// TIA Portal V20 export
DATA_BLOCK "Config"   // DB100
// stored: MemoryReserve 100, Namespace Unit1.Em7
   VAR
      em : "LAF_typeEmConfiguration";   // Configuration of EM Parameters
      axis : Array[1.._.U1EM7_NO_OF_AXES] of DB_ANY;
      cam : Array[1.._.U1EM7_NO_OF_AXES] of DB_ANY;
      moduleAccessPoint : Array[1.._.U1EM7_NO_OF_AXES] of HW_SUBMODULE;
   END_VAR
   VAR RETAIN
      cmNgKickerAxisZ : "LBC_typeAxisControlConfiguration";
      cmPassKickerAxisZ : "LBC_typeAxisControlConfiguration";
      cmCutConveyorAxisB : "LBC_typeAxisControlConfiguration";
      cmNgConveyorAxisB : "LBC_typeAxisControlConfiguration";
      cmStack1ConveyorAxisB : "LBC_typeAxisControlConfiguration";
      cmStack2ConveyorAxisB : "LBC_typeAxisControlConfiguration";
      cmConveyorVirtualAxisB : "LBC_typeAxisControlConfiguration";
      cmCutConveyorRingBlow : "LBC_typeSinaSpeedConfiguration";
      cmNgConveyorRingBlow : "LBC_typeSinaSpeedConfiguration";
      cmStack2ConveyorRingBlow : "LBC_typeSinaSpeedConfiguration";
      cmNgBoxLockCylinderUpDown : "LBC_typeTwoWayActuatorConfiguration";
      CmNgBoxDetectSensor : "LBC_typeDigitalSignalConfiguration";
      CmNgBoxFullSensor : "LBC_typeDigitalSignalConfiguration";
      CmNgKickerDetectSensor : "LBC_typeDigitalSignalConfiguration";
      CmPassKickerDetectSensor : "LBC_typeDigitalSignalConfiguration";
      CmStack1ConveyorElectrodeDetectSensor : "LBC_typeDigitalSignalConfiguration";
      CmStack2ConveyorElectrodeDetectSensor : "LBC_typeDigitalSignalConfiguration";
      cmStack1QrReader : "LER_typeSRX300Configuration";
      cmStack2QrReader : "LER_typeSRX300Configuration";
      cmNgKickerAxisZ_TorqueCal : "LER_typeServoTorqueCalConfigruation";
      cmPassKickerAxisZ_TorqueCal : "LER_typeServoTorqueCalConfigruation";
      cmCutConveyorAxisB_TorqueCal : "LER_typeServoTorqueCalConfigruation";
      cmNgConveyorAxisB_TorqueCal : "LER_typeServoTorqueCalConfigruation";
      cmStack1ConveyorAxisB_TorqueCal : "LER_typeServoTorqueCalConfigruation";
      cmStack2ConveyorAxisB_TorqueCal : "LER_typeServoTorqueCalConfigruation";
   END_VAR
BEGIN
   // axis[1] : cmNgKickerAxisZ
   // axis[2] : cmPassKickerAxisZ
   // axis[3] : cmCutConveyorAxisB
   // axis[4] : cmNgConveyorAxisB
   // axis[5] : cmStack1ConveyorAxisB
   // axis[6] : cmStack2ConveyorAxisB
   // axis[7] : cmCutConveyorRingBlow
   // axis[8] : cmNgConveyorRingBlow
   // axis[9] : cmStack2ConveyorRingBlow
   // axis[10] : cmConveyorVirtualAxisB
   // cam[1] : cmNgKickerAxisZ
   // cam[2] : cmPassKickerAxisZ
   // cam[3] : cmCutConveyorAxisB
   // cam[4] : cmNgConveyorAxisB
   // cam[5] : cmStack1ConveyorAxisB
   // cam[6] : cmStack2ConveyorAxisB
   // cam[7] : cmStack2ConveyorAxisB
   // cam[8] : cmNgConveyorRingBlow
   // cam[9] : cmStack2ConveyorRingBlow
   // cam[10] : cmConveyorVirtualAxisB
   // moduleAccessPoint[1] : cmNgKickerAxisZ
   // moduleAccessPoint[2] : cmPassKickerAxisZ
   // moduleAccessPoint[3] : cmCutConveyorAxisB
   // moduleAccessPoint[4] : cmNgConveyorAxisB
   // moduleAccessPoint[5] : cmStack1ConveyorAxisB
   // moduleAccessPoint[6] : cmStack2ConveyorAxisB
   // moduleAccessPoint[7] : cmCutConveyorRingBlow
   // moduleAccessPoint[8] : cmNgConveyorRingBlow
   // moduleAccessPoint[9] : cmStack2ConveyorRingBlow
   // moduleAccessPoint[10] : cmConveyorVirtualAxisB
   cmStack1QrReader.hwID.readDataExtendedPart1HwId := 530;
   cmStack1QrReader.hwID.readDataExtendedPart2HwId := 530;
   cmStack1QrReader.hwID.readDataExtendedPart3HwId := 530;
   cmStack2QrReader.hwID.readDataExtendedPart1HwId := 550;
   cmStack2QrReader.hwID.readDataExtendedPart2HwId := 550;
   cmStack2QrReader.hwID.readDataExtendedPart3HwId := 550;
END_DATA_BLOCK
